# B&R Automation Studio project EasyLog (part 2)

#### rtkMemory.h
```c
/**
 * @file
 * @brief RTK memory functions
 * @ingroup rtk
 */

#ifndef _RTK_MEMORY_H_
#define _RTK_MEMORY_H_

#include <rtkBase.h>

#ifdef __cplusplus
extern "C" {
#endif

/** @brief Type of RTK memory access flags */
typedef unsigned long RTK_MEMORY_ACCESS;

/** @name Memory access flags */
/*@{*/
#define RTK_MEM_NO_READ 0x00000000       /**< @brief ignored */
#define RTK_MEM_NO_WRITE 0x00000000      /**< @brief ignored */
#define RTK_MEM_NOT_EXECUTE 0x00000000   /**< @brief ignored */
#define RTK_MEM_READ_ALL 0x00000001      /**< @brief ignored */
#define RTK_MEM_WRITE_ALL 0x00000002     /**< @brief ignored */
#define RTK_MEM_EXECUTE_ALL 0x00000004   /**< @brief ignored */
#define RTK_MEM_READ_LOCAL 0x00000008    /**< @brief ignored */
#define RTK_MEM_WRITE_LOCAL 0x00000010   /**< @brief ignored */
#define RTK_MEM_EXECUTE_LOCAL 0x00000020 /**< @brief ignored */
#define RTK_MEM_NO_INIT 0x00000000       /**< @brief no memory initialization */
#define RTK_MEM_INITZERO 0x00008000      /**< @brief memory initialization with 0 */
/*@}*/

/**
 * @brief Allocates heap memory.
 *
 * Depending on the 'AccessFlags', the memory will be initialized with 0 (#RTK_MEM_INITZERO) or it will be not initialized
 * (#RTK_MEM_NO_INIT). After the function call 'lpMemoryAddress' (which must not be NULL) contains the pointer to the
 * allocated memory */
EXIMPORT RTK_ERROR RtkAllocateMemory(ULONG ulByteLength, RTK_MEMORY_ACCESS AccessFlags, void** lpMemoryAddress);

/**
 * @brief Frees memory allocated with RtkAllocateMemory().
 *
 * 'lpMemoryaddress' is the pointer to the memory to be freed */
EXIMPORT RTK_ERROR RtkFreeMemory(void* lpMemoryAddress, ULONG ulUnused);

/**
 * @brief Retrieves information about the DRAM
 * @param lpulMemSize              Output-parameter - can be NULL. Returns the overall RAM size in byte.
 * @param lpulFreeMemSize          Output-parameter - can be NULL. Returns the available/free RAM size in byte.
 * @param lpulBiggestFreeBlockSize Output-parameter - can be NULL. Returns the  biggest available/free consecutive
 *                                                              RAM block in byte. */
EXIMPORT RTK_ERROR RtkGetMemoryInfo(ULONG* lpulMemSize, ULONG* lpulFreeMemSize, ULONG* lpulBiggestFreeBlockSize);

#ifdef __cplusplus
}
#endif

#endif
```

#### rtkMisc.h
```c
/**
 * @file
 * @brief Miscellaneous RTK functions
 * @ingroup rtk
 */

#ifndef _RTK_MISC_H_
#define _RTK_MISC_H_

#include <rtkBase.h>

#ifdef __cplusplus
extern "C" {
#endif

/**
 * @brief Gets the current value of a microsecond counter.
 *
 * Can be used for time measurements.
 * Overflow from 0xFFFFFFFF to 0x00000000 */
EXIMPORT ULONG RtkReadUsecCounter(void);

/**
 * @brief Gets the configured system tick */
EXIMPORT ULONG RtkGetSystemTick(void);

#ifdef __cplusplus
}
#endif

#endif
```

#### arexport.h
```c
/**
 * @file
 * @brief This headerfile contains macros used to indicate the validity of exported functions.
 * @ingroup arsystem
 *
 */

#ifndef _AR_EXPORT_H_
#define _AR_EXPORT_H_

/**
 * @brief Functions marked with #AR_DEPRECATED should not be used in AR-external code at all.
 *
 * AR still supports these functions, but cannot provide guarantees for the compatibility
 * of these functions.
 * Any AR-external code using #AR_DEPRECATED functions should replace these functions with
 * the equivalent exported function which is not marked as #AR_DEPRECATED.
 */
#if !defined(AR_CORE) && defined(__GNUC__)
#define AR_DEPRECATED __attribute__((deprecated))
#else
#define AR_DEPRECATED
#endif

/**
 * @brief Functions marked with #AR_NOT_RECOMMENDED should not be used when writing new AR-external code.
 *
 * For these functions there is no functionally equivalent alternative available and thus
 * they cannot be replaced easily in existing code (that is why they are not #AR_DEPRECATED).
 */
#define AR_NOT_RECOMMENDED

#endif
```

### Program Logical/LoadCPU

#### Variables.var
```iecst
VAR
	TestBool : BOOL := FALSE;
	i : DINT := 0;
	NumberOfChanges : DINT := 1000;
END_VAR
```

#### Main.st
```iecst
PROGRAM _INIT
	(* Insert code here *)

END_PROGRAM

PROGRAM _CYCLIC
	(* Insert code here *)
	FOR i := 0 TO NumberOfChanges DO
		TestBool := NOT TestBool;

	END_FOR;
END_PROGRAM

PROGRAM _EXIT
	(* Insert code here *)

END_PROGRAM
```

### Program Logical/Program

#### Variables.var
```iecst
VAR
	ErrorNumberTest : UINT := 12345;
	LogMessageTest2 : STRING[256] := 'msg2';
	LogMessageTest : STRING[256] := 'msg1';
	LoggerName2 : STRING[20] := 'logger2';
	LoggerName : STRING[20] := 'logger1';
	InsertLog : BOOL;
	WriteLog : BOOL;
	Status1 : DINT;
	Status2 : DINT;
END_VAR
```

#### Main.st
```iecst
PROGRAM _INIT
	(* Insert code here *)

END_PROGRAM

PROGRAM _CYCLIC

	IF InsertLog THEN
		InsertLog := FALSE;
//		Objective, change the FB TO pass the Logger name instead OF the LogFifo
		UserLogEnqueue(arEVENTLOG_SEVERITY_ERROR, ErrorNumberTest,ADR(LogMessageTest),ADR(LoggerName));
		UserLogEnqueue(arEVENTLOG_SEVERITY_ERROR, ErrorNumberTest,ADR(LogMessageTest2),ADR(LoggerName2));

	END_IF;

		Status1 := UserLogWrite(ADR(LoggerName));
		Status2 := UserLogWrite(ADR(LoggerName2));

END_PROGRAM

PROGRAM _EXIT
	(* Insert code here *)

END_PROGRAM
```

Listed in the project but not available here: Logical/Global.typ, Logical/Global.var, Logical/Libraries/EasyLog/AsyncCreation/ARM/rtkSemaphore.h, Logical/Libraries/EasyLog/AsyncCreation/ARM/rtkSharedMemory.h, Logical/Libraries/EasyLog/AsyncCreation/ARM/rtkTask.h, Logical/Libraries/EasyLog/AsyncCreation/ARM/rtkTimer.h, Logical/Libraries/EasyLog/AsyncCreation/ARM/rtkTypes.h, Logical/Libraries/EasyLog/AsyncCreation/ARM/rLib.h, Logical/Libraries/EasyLog/AsyncCreation/ARM/rtk.h, Logical/Libraries/EasyLog/AsyncCreation/ARM/rtkBase.h, Logical/Libraries/EasyLog/AsyncCreation/ARM/rtkCriticalSection.h, Logical/Libraries/EasyLog/AsyncCreation/ARM/rtkFifo.h, Logical/Libraries/EasyLog/AsyncCreation/ARM/rtkInterrupt.h, Logical/Libraries/EasyLog/AsyncCreation/ARM/rtkMemory.h, Logical/Libraries/EasyLog/AsyncCreation/ARM/rtkMisc.h, Logical/Libraries/EasyLog/AsyncCreation/ARM/rtkObject.h, Logical/Libraries/EasyLog/AsyncCreation/ARM/rtkPlainFifo.h, Logical/Libraries/EasyLog/AsyncCreation/ARM/arexport.h, Logical/Async/AsyncTask/Types.typ, Logical/FunAsync/Init.c, Logical/FunAsync/Exit.c, Logical/FunAsync/Types.typ, Logical/FunAsync/_inc/rtkRtc.h, Logical/FunAsync/_inc/rtkTask.h, Logical/FunAsync/_inc/rtkTimer.h, Logical/FunAsync/_inc/rtkTypes.h, Logical/FunAsync/_inc/rtk.h, Logical/FunAsync/_lib/_IA32
